(* IEC 61131-3 sources: cc_kush_rewrite/Functions/Sensors, 7 files *)

(* ---- FC_Sensor_CheckGS.st ---- *)
FUNCTION FC_Sensor_CheckGS : BOOL
VAR_INPUT
	fbGS : REFERENCE TO FB_UniversalSignal;
END_VAR
VAR
END_VAR
// Контроль заштыбовки (1 - норма, 0 - заштыбовка)
FC_Sensor_CheckGS := NOT fbGS.qxSignal;

END_FUNCTION

(* ---- FC_Sensor_CheckHQ.st ---- *)
FUNCTION FC_Sensor_CheckHQ : BOOL
VAR_INPUT
	fbHQ_IsOk : REFERENCE TO ARRAY[1..4] OF FB_UniversalSignal;
END_VAR
VAR
END_VAR
// Кабель-тросовый выключатель (1 - норма, 0 - стоп)
FC_Sensor_CheckHQ := (
	NOT fbHQ_IsOk[1].qxSignal
	OR NOT fbHQ_IsOk[2].qxSignal
	OR NOT fbHQ_IsOk[3].qxSignal
	OR NOT fbHQ_IsOk[4].qxSignal
);

END_FUNCTION

(* ---- FC_Sensor_CheckSQ.st ---- *)
FUNCTION FC_Sensor_CheckSQ : BOOL
VAR_INPUT
	fbSQ_IsOk : REFERENCE TO ARRAY[1..2] OF FB_UniversalSignal;
END_VAR
VAR
END_VAR
// Контроль ограждения барабана (1 - норма, 0 - ограждения нет)
FC_Sensor_CheckSQ := (
	NOT fbSQ_IsOk[1].qxSignal
	OR NOT fbSQ_IsOk[2].qxSignal
);

END_FUNCTION

(* ---- FC_Sensor_CheckYE.st ---- *)
FUNCTION FC_Sensor_CheckYE : BOOL
VAR_INPUT
	fbYE : REFERENCE TO FB_UniversalSignal;
END_VAR
VAR
END_VAR
// Обнаружение металла (1 - обнаружение, 0 - нет)
FC_Sensor_CheckYE := fbYE.qxSignal;

END_FUNCTION

(* ---- FC_Sensor_CheckYS.st ---- *)
FUNCTION FC_Sensor_CheckYS : BOOL
VAR_INPUT
	fbYS : REFERENCE TO FB_UniversalSignal;
END_VAR
VAR
END_VAR
// Контроль продольного разрыва ленты (1 - норма, 0 - разрыв)
FC_Sensor_CheckYS := NOT fbYS.qxSignal;

END_FUNCTION

(* ---- FC_Sensor_CheckZQAlarm.st ---- *)
FUNCTION FC_Sensor_CheckZQAlarm : BOOL
VAR_INPUT
	fbZQAlarm : REFERENCE TO ARRAY[1..4] OF FB_UniversalSignal;
END_VAR
VAR
END_VAR
// Контроль схода ленты - тревога (1 - норма, 0 - стоп)
FC_Sensor_CheckZQAlarm := (
	NOT fbZQAlarm[1].qxSignal
	OR NOT fbZQAlarm[2].qxSignal
	OR NOT fbZQAlarm[3].qxSignal
	OR NOT fbZQAlarm[4].qxSignal
);

END_FUNCTION

(* ---- FC_Sensor_CheckZQWarning.st ---- *)
FUNCTION FC_Sensor_CheckZQWarning : BOOL
VAR_INPUT
	fbZQWarning : REFERENCE TO ARRAY[1..4] OF FB_UniversalSignal;
END_VAR
VAR
END_VAR
// Контроль схода ленты - тревога (1 - норма, 0 - стоп)
FC_Sensor_CheckZQWarning := (
	NOT fbZQWarning[1].qxSignal
	OR NOT fbZQWarning[2].qxSignal
	OR NOT fbZQWarning[3].qxSignal
	OR NOT fbZQWarning[4].qxSignal
);

END_FUNCTION
